TYPE ST185_PnpHorPos_e : ST110_PnpHorPos_e;
END_TYPE

(* stored: Version 1.1.0.1, ProductVersion 3.1.4024.6
   DUT ST185_PnpHorPos_e: Id {8d366203-8902-4fe9-b296-5180a1ad09c3} *)
